{attribute 'call_after_init'}
FUNCTION_BLOCK FB_DumpChillerEnable_Test EXTENDS FB_TestSuite
VAR_INPUT
END_VAR
VAR_OUTPUT
END_VAR
VAR
END_VAR

LocksWithHardwareFailure();
LocksWithLUTLeak();
LocksWithLOTAOLeak();
LocksWithLOTNLLeak();
LocksWithLOCOLeak();
EnablesWhenNoError();

METHOD EnablesWhenNoError
VAR
	stErrors : st_ErrorStates;
	bResult : BOOL;
END_VAR
TEST('EnablesWhenNoError');

bResult := F_DumpChillerEnable(stErrors := stErrors);

AssertTrue(bResult, 'Dump chiller relay did not close');

TEST_FINISHED();
END_METHOD

METHOD LocksWithHardwareFailure
VAR
	stErrors : st_ErrorStates;
	bResult : BOOL;
END_VAR
TEST('LocksWithHardwareFailure');

stErrors.bHardwareFailure := TRUE;
bResult := F_DumpChillerEnable(stErrors := stErrors);

AssertFalse(bResult, 'Dump chiller relay did not open');

TEST_FINISHED();
END_METHOD

METHOD LocksWithLOCOLeak
VAR
	stErrors : st_ErrorStates;
	bResult : BOOL;
END_VAR
TEST('LocksWithLOCOLeak');

stErrors.bLeakOpcpaCarbideOn := TRUE;
bResult := F_DumpChillerEnable(stErrors := stErrors);

AssertFalse(bResult, 'Dump chiller relay did not open');

TEST_FINISHED();
END_METHOD

METHOD LocksWithLOTAOLeak
VAR
	stErrors : st_ErrorStates;
	bResult : BOOL;
END_VAR
TEST('LocksWithLOTAOLeak');

stErrors.bLeakOpticalTableAmphosOn := TRUE;
bResult := F_DumpChillerEnable(stErrors := stErrors);

AssertFalse(bResult, 'Dump chiller relay did not open');

TEST_FINISHED();
END_METHOD

METHOD LocksWithLOTNLLeak
VAR
	stErrors : st_ErrorStates;
	bResult : BOOL;
END_VAR
TEST('LocksWithLOTNLLeak');

stErrors.bLeakOpticalTableNoLaser := TRUE;
bResult := F_DumpChillerEnable(stErrors := stErrors);

AssertFalse(bResult, 'Dump chiller relay did not open');

TEST_FINISHED();
END_METHOD

METHOD LocksWithLUTLeak
VAR
	stErrors : st_ErrorStates;
	bResult : BOOL;
END_VAR
TEST('LocksWithLUTLeak');

stErrors.bLeakUnderTable := TRUE;
bResult := F_DumpChillerEnable(stErrors := stErrors);

AssertFalse(bResult, 'Dump chiller relay did not open');

TEST_FINISHED();
END_METHOD

END_FUNCTION_BLOCK

(* stored: Version 1.1.0.1, ProductVersion 3.1.4022.17
   POU FB_DumpChillerEnable_Test: Id {a14a40e3-e678-4c74-b00e-5f2ba0622eed}, SpecialFunc None
   Method EnablesWhenNoError: Id {85dda632-467c-4749-a511-cdb805b38063}
   Method LocksWithHardwareFailure: Id {4305fef1-3f26-4339-8562-d40fb551ab84}
   Method LocksWithLOCOLeak: Id {2e88444b-c045-4dc5-bbd8-8671c9554878}
   Method LocksWithLOTAOLeak: Id {e53b8efc-a6a2-4f5f-b303-4716304d0f05}
   Method LocksWithLOTNLLeak: Id {1f7a6d3d-be09-417b-8842-c43116a9599b}
   Method LocksWithLUTLeak: Id {7dfde73b-deb2-4b0f-a5b0-be5e5c1041dd} *)
